ABB RobotStudio station: dual_20220310-134731.rsstn

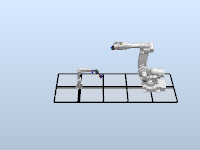
Station Station (saved by RobotStudio 21.4.9700.0)
Controller Dual_controller
  mechanical unit ROB_1: IRB1200_5_90_STD_03, 6 joints, base frame (0, 0, 0) mm
  mechanical unit ROB_2: IRB6640_180_255__04, 6 joints, base frame (3000, 0, 0) mm, rotated rx 0 ry 0 rz 180 deg
Layout (positions relative to the parent item):
  - IRB1200_5_90_STD_03 [mechanism, from Robots\IRB1200_5_90_STD_03.rslib] at (0, 0, 0) mm; joint values [0, 0, 0, 0, 0.5236, 0] (rad or m)
  - IRB6640_180_255__04 [mechanism, from Robots\IRB6640_180_255_G_04.rslib] at (3000, 0, 0) mm, rotated rx 0 ry 0 rz 180 deg; joint values [0, 0, 0, 0, 0.5236, 0] (rad or m)
  - MyNewTool [mechanism, from models\Paintgun.rslib] at (522.01, 0, 848.1) mm, rotated rx 180 ry 60 rz 180 deg
Attachment: MyNewTool is attached to IRB1200_5_90_STD_03 / Link6
Targets, tools, work objects and paths stored in the station, written as RAPID:
! task T_ROB1
MODULE CalibData
  PERS tooldata MyNewTool:=[TRUE,[[50,0,450],[1,0,0,0]],[1,[0,0,1],[1,0,0,0],0,0,0]];
ENDMODULE

